FUNCTION_BLOCK ABSTRACT HaltedProgramState EXTENDS ProgramState

{attribute 'monitoring' := 'call'}
{attribute 'OPC.UA.DA.Property' := '1'}
{attribute 'OPC.UA.DA.Access' := '1'}
PROPERTY FINAL Name : STRING
GET
Name := 'Halted';
END_GET
END_PROPERTY

END_FUNCTION_BLOCK

(* stored: Version 1.1.0.1
   POU HaltedProgramState: Id {a9eee460-5125-4d00-bef3-ce2985ca3212}, SpecialFunc None
   Property Name: Id {b967a08b-8ec4-45ba-b5b7-013ea0ce9029}
   Get Get: Id {4c0e5d56-7101-4ea9-9d8c-2247c5aebe86} *)
